// SIMATIC S7-200 project (STEP 7-Micro/WIN), CPU 221 REL 01.10

ORGANIZATION_BLOCK 主程序:OB1
TITLE=程序注释
BEGIN
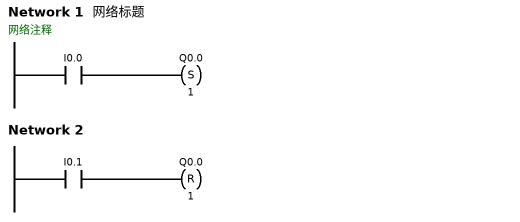
Network 1 // 网络标题
// 网络注释
LD     I0.0
S      Q0.0, 1
Network 2
LD     I0.1
R      Q0.0, 1
END_ORGANIZATION_BLOCK
